// Mitsubishi GX Works2 project: TH05   PLC: FX2N/FX2NC

PROGRAM MAIN
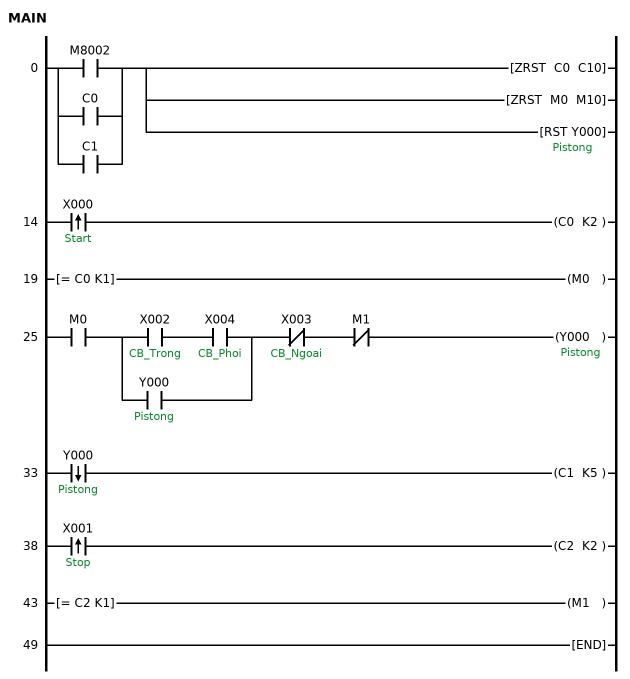
0     LD      M8002
      OR      C0
      OR      C1
      ZRST    C0 C10
      ZRST    M0 M10
      RST     Y000  ; Pistong
14    LDP     X000  ; Start
      OUT     C0 K2
19    LD=     C0 K1
      OUT     M0
25    LD      M0
      LD      X002  ; CB_Trong
      AND     X004  ; CB_Phoi
      OR      Y000  ; Pistong
      ANB
      ANI     X003  ; CB_Ngoai
      ANI     M1
      OUT     Y000  ; Pistong
33    LDF     Y000  ; Pistong
      OUT     C1 K5
38    LDP     X001  ; Stop
      OUT     C2 K2
43    LD=     C2 K1
      OUT     M1
49    END
END_PROGRAM
